// TIA Portal V17 export
// export: Created 2024-08-07T21:44:11.0411207Z, ExportSetting WithDefaults, DisplayName Totally Integrated Automation Portal, DisplayVersion V17 Update 7, DisplayName TIA Portal Openness, DisplayVersion V17 Update 7, DisplayName TIA Portal Version Control Interface, DisplayVersion V17, DisplayName SINAMICS Startdrive Advanced, DisplayVersion V17 SP2, DisplayName SINAMICS Startdrive G110M, G120, G120C, G120D, G120P, G115D, DisplayVersion V17 SP2, DisplayName SINAMICS Startdrive G130, G150, S120, S150, SINAMICS MV, S210, DisplayVersion V17 SP2, DisplayName STEP 7 Professional, DisplayVersion V17 Update 7, DisplayName STEP 7 Safety, DisplayVersion V17 Update 6, DisplayName WinCC Advanced / Unified PC, DisplayVersion V17 Update 7
FUNCTION_BLOCK "7. Call_M103_PY"   // FB2007, LAD
{ S7_Optimized_Access := 'TRUE' }
VERSION : 0.1
// stored: AutoNumber false, IsIECCheckEnabled false, IsRetainMemResEnabled false, MemoryReserve 100, SetENOAutomatically false, UDAEnableTagReadback false
   VAR_INPUT
      PY_ON { ExternalAccessible := 'False'; ExternalVisible := 'False'; ExternalWritable := 'False'} : Bool;
      PY_DOWN { ExternalAccessible := 'False'; ExternalVisible := 'False'; ExternalWritable := 'False'} : Bool;
      PY_OFF { ExternalAccessible := 'False'; ExternalVisible := 'False'; ExternalWritable := 'False'} : Bool;
   END_VAR
   VAR
      PYOnTemp : Bool;
      PYDownTemp : Bool;
      PYOffTemp : Bool;
   END_VAR
BEGIN

REGION Network 1 (SCL)
   IF (#PY_ON <> #PYOnTemp OR #PY_DOWN <> #PYDownTemp OR #PY_OFF <> #PYOffTemp) AND (#PY_ON OR #PY_DOWN OR #PY_OFF) THEN

       "MII_Interface_Data".MII_METHODS.M103_PY.Inputs.PLC_ID := "MII_Parameters".Connection.PLC_ID;
       "MII_Interface_Data".MII_METHODS.M103_PY.Inputs.PLANT := "MII_Parameters".Connection.PlantID;

       "MII_Interface_Data".MII_METHODS.M103_PY.Inputs.PY_ON := #PY_ON;
       "MII_Interface_Data".MII_METHODS.M103_PY.Inputs.PY_DOWN := #PY_DOWN;
       "MII_Interface_Data".MII_METHODS.M103_PY.Inputs.PY_OFF := #PY_OFF;

       //Call the method 
       "1. DMC_setConnection_DB".CallBuffer[7] := TRUE;

       #PYOnTemp := #PY_ON;
       #PYDownTemp := #PY_DOWN;
       #PYOffTemp := #PY_OFF;
   END_IF;
END_REGION
END_FUNCTION_BLOCK
